PROGRAM SouthLight_Control
VAR
	StraightGreenLight  : BOOL := FALSE;	//Controls if the green light is on
	StraightYellowLight : BOOL := FALSE;	//Controls if the yellow light is on
	StraightRedLight    : BOOL := TRUE; 	//Controls if the red light is on
	
	StraightOnTimer : INT := 0;				//Tracks how long the light has been on
	
	LeftGreenLight  : BOOL := FALSE;		//Controls if the green light is on
	LeftYellowLight : BOOL := FALSE;		//Controls if the yellow light is on
	leftRedLight    : BOOL := TRUE; 		//Controls if the red light is on
	
	LeftOnTimer : INT := 0;					//Tracks how long the light has been on
	
	CrosswalkLight : BOOL := FALSE;			//Controls if the crosswalk light is on (walk=TRUE)
END_VAR

//If all of the sensors and lights are off, default to N/S straight
IF Glbl.northStraightSensor = FALSE AND  Glbl.northLeftSensor = FALSE AND Glbl.southStraightSensor = FALSE AND Glbl.southLeftSensor = FALSE AND Glbl.eastStraightSensor = FALSE AND Glbl.eastLeftSensor = FALSE AND Glbl.westStraightSensor = FALSE AND Glbl.westLeftSensor = FALSE AND  Glbl.northLeftActive = FALSE AND Glbl.southLeftActive = FALSE AND Glbl.eastStraightActive = FALSE AND Glbl.eastLeftActive = FALSE AND Glbl.westStraightActive = FALSE AND Glbl.westLeftActive = FALSE THEN
	Glbl.southStraightActive := TRUE;
	StraightRedLight := FALSE;
	StraightGreenLight := TRUE;
ELSE //Control for the straight light if active
IF Glbl.southStraightActive = TRUE THEN			//If the straight light is set to be active
		IF StraightOnTimer = 0 THEN					//Take off half of the state counter when the light is activated
			//Glbl.state1Counter := Glbl.state1Counter - (Glbl.state1Counter/2);
			//Glbl.state6Counter := Glbl.state6Counter - (Glbl.state6Counter/2);		
		END_IF
		IF StraightOnTimer <= 10 THEN				//If the light has been on for 10 seconds or less, make it green
			StraightGreenLight := TRUE;
			StraightYellowLight := FALSE;
			StraightRedLight := FALSE;
			StraightOnTimer := StraightOnTimer + 1;	//Incriment the amount of time it has been on by 1
			Glbl.southStraightSensor := FALSE;		//Set the sensor to false
			Glbl.southStraightSensorCnt := MAX(Glbl.southStraightSensorCnt-1, 0);		//Set the car counter to 0
		ELSIF StraightOnTimer <= 13 THEN			//If the light has been on for 11-13 seconds, make it yellow
			StraightGreenLight := FALSE;
			StraightYellowLight := TRUE;
			StraightRedLight := FALSE;
			StraightOnTimer := StraightOnTimer + 1;	//Incriment the amount of time it has been on by 1
		ELSE										//Once it is done, turn it to red and set it as inactive, reset timer to 0
			StraightGreenLight := FALSE;
			StraightYellowLight := FALSE;
			StraightRedLight := TRUE;
			Glbl.southStraightActive := FALSE;
			StraightOnTimer := 0;	
		END_IF
	END_IF
END_IF

//Control for the left light if active
IF Glbl.southLeftActive = TRUE THEN			//If the left light is set to be active
	IF LeftOnTimer = 0 THEN					//Take off half of the state counter when the light is activated
		//Glbl.state3Counter := Glbl.state3Counter - (Glbl.state3Counter/2);
		//Glbl.state6Counter := Glbl.state6Counter - (Glbl.state6Counter/2);	
	END_IF
	IF LeftOnTimer <= 10 THEN				//If the light has been on for 10 seconds or less, make it green
		LeftGreenLight := TRUE;
		LeftYellowLight := FALSE;
		LeftRedLight := FALSE;
		LeftOnTimer := LeftOnTimer + 1;	//Incriment the amount of time it has been on by 1
		Glbl.southLeftSensor := FALSE; 		//Set the sensor to false
		Glbl.southLeftSensorCnt := MAX(Glbl.southLeftSensorCnt-1, 0);		//Set the car counter to 0
	ELSIF LeftOnTimer <= 13 THEN			//If the light has been on for 11-13 seconds, make it yellow
		LeftGreenLight := FALSE;
		LeftYellowLight := TRUE;
		LeftRedLight := FALSE;
		LeftOnTimer := LeftOnTimer + 1;	//Incriment the amount of time it has been on by 1
	ELSE									//Once it is done, turn it to red and set it as inactive, reset timer to 0
		LeftGreenLight := FALSE;
		LeftYellowLight := FALSE;
		LeftRedLight := TRUE;
		Glbl.southLeftActive := FALSE;
		LeftOnTimer := 0;	
	END_IF
END_IF

//If the sensor is on and the light is off, incirment the waiting counters
IF Glbl.southStraightSensor = TRUE AND Glbl.southStraightActive = FALSE THEN
	Glbl.state1Counter := Glbl.state1Counter + Glbl.southStraightSensorCnt;
	Glbl.state6Counter := Glbl.state6Counter + Glbl.southStraightSensorCnt;
END_IF
IF Glbl.southLeftSensor = TRUE AND Glbl.southLeftActive = FALSE THEN
	Glbl.state3Counter := Glbl.state3Counter + Glbl.southLeftSensorCnt;
	Glbl.state6Counter := Glbl.state6Counter + Glbl.southLeftSensorCnt;
END_IF

//Check to see if the crosswalk can be turned on
IF (Glbl.eastStraightActive = TRUE AND Glbl.westStraightActive = TRUE) OR (Glbl.westStraightActive = TRUE AND Glbl.westLeftActive = TRUE) THEN
	CrosswalkLight := TRUE;
ELSE
	CrosswalkLight := FALSE;
END_IF

END_PROGRAM

(* stored: Version 1.1.0.1, ProductVersion 3.1.4022.10
   POU SouthLight_Control: Id {4cbb6711-6eed-4d45-983d-a2f73b62deca}, SpecialFunc None *)
